{attribute 'TcGenerated'}
{attribute 'no-analysis'}
{attribute 'linkalways'}
// This function has been automatically generated from the project information.
VAR_GLOBAL CONSTANT
    {attribute 'const_non_replaced'}
    stLibVersion_qrix_motion : ST_LibVersion := (iMajor := 0, iMinor := 3, iBuild := 0, iRevision := 0, nFlags := 1, sVersion := '0.3.0');
END_VAR

(* stored: Version 1.1.0.1, ProductVersion 3.1.4022.18
   GVL Global_Version: Id {59aeb031-1144-48c9-bd4a-a8d497dc3ac8} *)
